PROGRAM MAIN
VAR
END_VAR

END_PROGRAM

(* stored: Version 1.1.0.1
   POU MAIN: Id {eff31504-fe48-4848-9ae3-b9f0c0832f2c} *)
